// TIA Portal V21 export
DATA_BLOCK "PRINT DATA"   // DB39
{ S7_Optimized_Access := 'FALSE' }
   VAR RETAIN
      "PRINT INTERVAL" : Int := 0;
      "PRODUCT NAME" : String := '';
      "BATCH NO" : String := '';
      "OPERATOR NAME" : String := 'UDAYLAL';
      "RECIPE TYPE" : String := '  ';
      "EQUIPMENT ID" : String := 'C1/A/INJ/AUT-05';
      "TUNNEL MODE" : String := 'STANDARD3 CYCLE SELECTED';
      "BATCH SIZE" : String := '0488';
      "CONTAINER NO" : String := '';
      NEW : String := '';
      QUANTITY : String;
   END_VAR
BEGIN
END_DATA_BLOCK
